RoboDK station: ROBODK_SIGNAL_BOX_V1.rdk

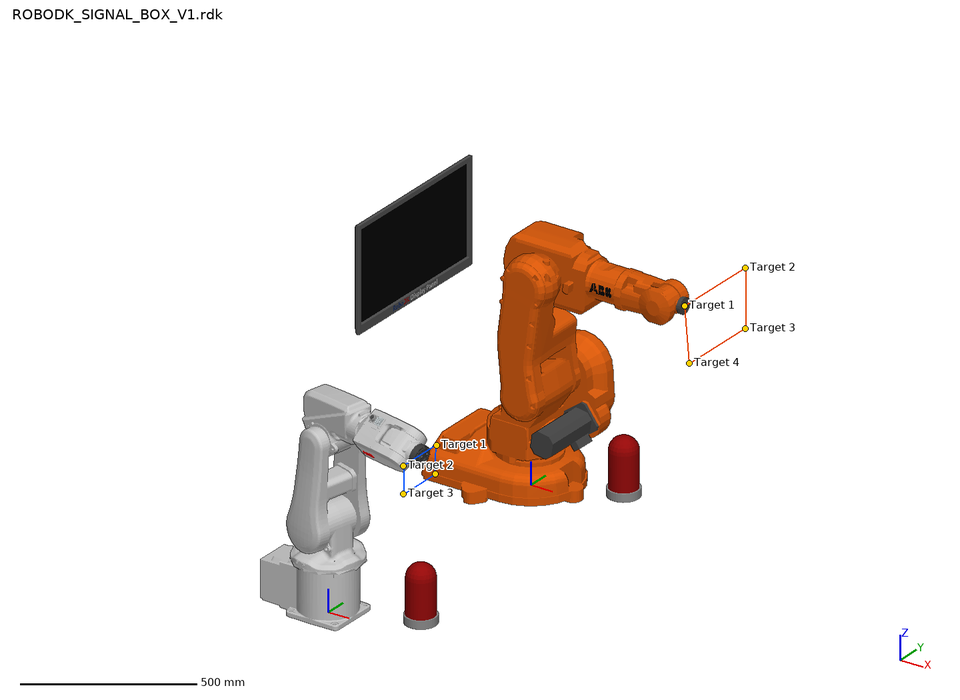
[picture v0: the station drawn from its stored meshes, robots at their saved joint values, targets as dots, program paths as lines]
Station ROBODK 3D PRINT AND CONTROLLER (saved by RoboDK 5.7.4). Poses are relative to the parent item; angles as X-Y-Z fixed-axis rotations.
Station parameters (name, value as stored): IO_1, 0, IO_2, 0, Photodiode, 740
  - frame ABB IRB 120-3/0.6 Base at (0, 0, 0) mm
    - robot ABB IRB 120-3/0.3 (model ABB IRB 120-3/0.6): 6 axes, payload 3 kg, reach 580 mm, repeatability 0.01 mm, weight 25 kg
        modified DH rows (alpha deg, a mm, theta deg, d mm): 0, 0, 0, 290; -90, 0, -90, 0; 0, 270, 0, 0; -90, 70, 0, 302; 90, 0, 0, 0; -90, 0, 180, 72
        joint limits [-165, -110, -90, -160, -120, -400] to [165, 110, 70, 160, 120, 400]; home [0, 0, 0, 0, 0, 0]; saved at [-12.428, 3.919, -4.192, 38.932, 12.431, -38.863]
    - target Target 1 (Cartesian target) at (374, 0, 630) mm, rotated rx 0 ry 90 rz 0 deg; joints [0, 0, 0, 0, 0, 0] of ABB IRB 120-3/0.3
    - target Target 2 (Cartesian target) at (374, -163.03, 630) mm, rotated rx 0 ry 90 rz 0 deg; joints [-28.361, 8.943, -9.567, 88.845, 28.367, -88.688] of ABB IRB 120-3/0.3
    - target Target 3 (Cartesian target) at (374, -163.03, 540.71) mm, rotated rx 0 ry 90 rz 0 deg; joints [-28.361, 7.162, 9.065, 117.369, 32.337, -121.495] of ABB IRB 120-3/0.3
    - target Target 4 (Cartesian target) at (374, -6.94, 540.71) mm, rotated rx 0 ry 90 rz 0 deg; joints [-1.317, -1.556, 18.155, -4.601, -16.65, 4.409] of ABB IRB 120-3/0.3
  - frame ABB IRB 140-6/0.8 Base at (0, 1000, 0) mm
    - robot ABB IRB 140-6/0.8: 6 axes, payload 6 kg, reach 810 mm, repeatability 0.03 mm, weight 98 kg
        modified DH rows (alpha deg, a mm, theta deg, d mm): 0, 0, 0, 352; -90, 70, -90, 0; 0, 360, 0, 0; -90, 0, 0, 380; 90, 0, 0, 0; -90, 0, 180, 65
        joint limits [-180, -90, -230, -200, -120, -400] to [180, 110, 50, 200, 120, 400]; home [0, 0, 0, 0, 0, 0]; saved at [0, 2.547, -2.601, 0, 0.054, 0]
    - target Target 1 (Cartesian target) at (531, 0, 712) mm, rotated rx 0 ry 90 rz 0 deg; joints [0, 2.547, -2.601, 0, 0.054, 0] of ABB IRB 140-6/0.8
    - target Target 2 (Cartesian target) at (531, 299.55, 712) mm, rotated rx 0 ry 90 rz 0 deg; joints [32.733, 16.839, -19.167, -86.384, 32.807, 85.7] of ABB IRB 140-6/0.8
    - target Target 3 (Cartesian target) at (531, 299.55, 521.32) mm, rotated rx 0 ry 90 rz 0 deg; joints [32.733, 22.942, 2.325, -123.585, 40.473, 131.118] of ABB IRB 140-6/0.8
    - target Target 4 (Cartesian target) at (531, 23.54, 521.32) mm, rotated rx 0 ry 90 rz 0 deg; joints [2.892, 10.334, 18.771, -174.07, 29.236, 174.821] of ABB IRB 140-6/0.8
  - program Start rob 1 (7 instructions, listed below)
  - program Start rob 2 (7 instructions, listed below)
  - program SET_IO1_0 (3 instructions, listed below)
  - program SET_IO1_1 (4 instructions, listed below)
  - program SET_IO2_0 (3 instructions, listed below)
  - program SET_IO2_1 (4 instructions, listed below)
  - program SET_PD (1 instructions, listed below)
  - object Light_R1_RED at (250, 100, 0) mm, size 100 x 100 x 185.3 mm, geometry from Light-Red.sld
  - object Light_R2_RED at (250, 1100, 0) mm, size 100 x 100 x 185.3 mm, geometry from Light-Red.sld
  - object Light_R1_GREEN at (250, 100, 0) mm, size 100 x 100 x 185.3 mm, geometry from Light-Red.sld
  - object Light_R2_GREEN at (250, 1100, 0) mm, size 100 x 100 x 185.3 mm, geometry from Light-Red.sld
  - object Display Panel 24in at (0, 400, 1000) mm, size 43 x 556.4 x 342.2 mm, geometry from PLUGIN_DISPLAY_DATAU
  - Python program serial_com_test_1 (listed below)
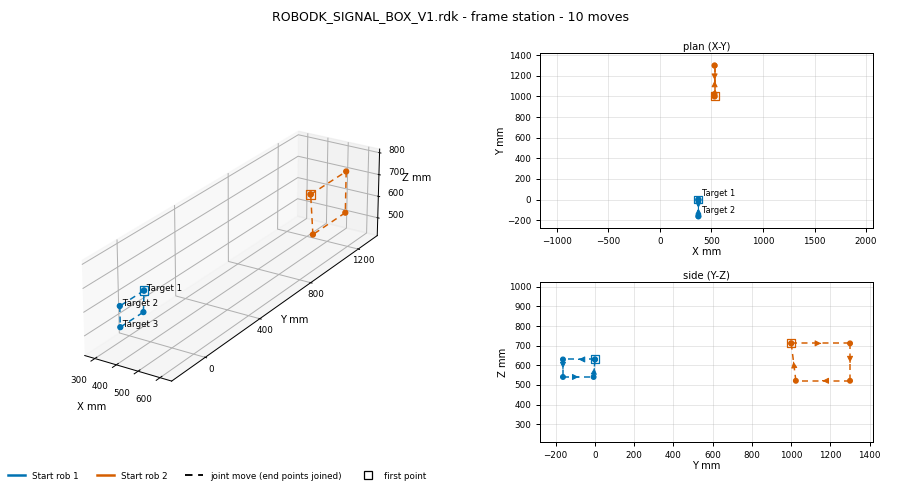
[picture p0: tool path of ROBODK_SIGNAL_BOX_V1.rdk in frame station, 10 of 10 moves have a stored position in this frame; points joined in program order, loops and branches not executed]

--- program Start rob 1 (robot ABB IRB 120-3/0.3) ---
  Set Ref.: ABB IRB 120-3/0.6 Base
  Wait IO_1=1
  MoveJ (Target 1)
  MoveJ (Target 2)
  MoveJ (Target 3)
  MoveJ (Target 4)
  MoveJ (Target 1)

--- program Start rob 2 (robot ABB IRB 140-6/0.8) ---
  Set Ref.: ABB IRB 140-6/0.8 Base
  Wait IO_2=1
  MoveJ (Target 1)
  MoveJ (Target 2)
  MoveJ (Target 3)
  MoveJ (Target 4)
  MoveJ (Target 1)

--- program SET_IO1_0 (robot ABB IRB 120-3/0.3) ---
  Set IO_1=0
  Hide Light_R1_GREEN
  Show Light_R1_RED

--- program SET_IO1_1 (robot ABB IRB 120-3/0.3) ---
  Set IO_1=1
  Show Light_R1_GREEN
  Hide Light_R1_RED
  Call Start rob 1

--- program SET_IO2_0 (robot ABB IRB 120-3/0.3) ---
  Set IO_2=0
  Hide Light_R2_GREEN
  Show Light_R2_RED

--- program SET_IO2_1 (robot ABB IRB 120-3/0.3) ---
  Set IO_2=1
  Hide Light_R2_RED
  Show Light_R2_GREEN
  Call Start rob 2

--- program SET_PD (robot ABB IRB 120-3/0.3) ---
  Set AO_5=1

--- Python program serial_com_test_1 ---
import tkinter as tk
import time
import serial
from robolink import Robolink  # Ensure this is imported correctly
from datetime import datetime  # Import datetime module for formatting the timestamp

# Initialize RoboDK and serial communication
RDK = Robolink()
ser = serial.Serial('COM4', 115200)

# Keep track of previous sensor values
prev_sensor1_value = None
prev_sensor2_value = None

# Log file setup
log_file = "D:/UPB/2024_2025_SEM_1/Articole/01_RoboDK signal Box/documente_articol_v1/latency_log.txt"

# Function to log latency and timestamp
def log_latency(latency, timestamp):
    # Convert timestamp to a readable format
    formatted_time = datetime.fromtimestamp(timestamp).strftime('%Y-%m-%d %H:%M:%S.%f')
    with open(log_file, "a") as file:
        file.write(f"{formatted_time}, {latency:.6f} ms\n")

# Function to handle executing RoboDK programs and updating the UI label
def execute_program_and_update_label(program_name, label):
    RDK.RunProgram(program_name)
    if program_name == "SET_IO1_0":
        label["text"] = "Sensor 1 Value: 0"
        label["bg"] = "yellow"
    elif program_name == "SET_IO1_1":
        label["text"] = "Sensor 1 Value: 1"
        label["bg"] = "green"
    elif program_name == "SET_IO2_0":
        label["text"] = "Sensor 2 Value: 0"
        label["bg"] = "yellow"
    elif program_name == "SET_IO2_1":
        label["text"] = "Sensor 2 Value: 1"
        label["bg"] = "green"

# Function to continuously read data from Arduino and update the UI
def read_arduino_data():
    global prev_sensor1_value, prev_sensor2_value
    while True:
        try:
            # Flush the serial buffer if it's too full
            if ser.in_waiting > 100:
                ser.reset_input_buffer()

            # Start measuring time when data is read
            start_time_pc = time.perf_counter()

            # Read data from Arduino
            if ser.in_waiting > 0:
                data = ser.readline().decode().strip()

                # Split the data into sensor identifier, value, and timestamp
                sensor, value, arduino_timestamp = data.split('_')
                arduino_timestamp = float(arduino_timestamp)

                # Check the current mode (manual/automatic)
                if current_mode.get() == 1:  # Only process Arduino data in automatic mode
                    # Calculate processing time
                    processing_time = (time.perf_counter() - start_time_pc) * 1000  # Convert to ms

                    # Handle IO1 (sensor 1)
                    if sensor == "IO1" and value != prev_sensor1_value:
                        prev_sensor1_value = value
                        execute_program_and_update_label(f"SET_IO1_{value}", label_signal_s1)
                        print(f"Arduino-to-Python processing time: {processing_time:.6f} ms")

                    # Handle IO2 (sensor 2)
                    elif sensor == "IO2" and value != prev_sensor2_value:
                        prev_sensor2_value = value
                        execute_program_and_update_label(f"SET_IO2_{value}", label_signal_s2)
                        print(f"Arduino-to-Python processing time: {processing_time:.6f} ms")

                    # Handle Photodiode (PD) sensor
                    elif sensor == "PD":
                        label_signal_pd["text"] = f"Photodiode Value: {value}"
                        RDK.setParam('Photodiode', value)

                    # End measuring time after running the RoboDK program
                    end_time_pc = time.perf_counter()
                    end_to_end_latency = (end_time_pc - start_time_pc) * 1000  # Convert to ms
                    timestamp = time.time()  # Get the current time in seconds
                    print(f"End-to-End Latency: {end_to_end_latency:.6f} ms")

                     # Log the end-to-end latency and timestamp
                    log_latency(end_to_end_latency, timestamp)

            # Small delay to avoid overwhelming the buffer
            time.sleep(0.01)

        except Exception as e:
            print(f"Error reading Arduino data: {e}")

# Function to handle mode change in the UI (manual/automatic mode)
def change_mode():
    if current_mode.get() == 0:
        label_mode.config(text="Mode: Manual")
        for button in buttons_manual.values():
            button.config(state=tk.NORMAL)
    else:
        label_mode.config(text="Mode: Automatic")
        for button in buttons_manual.values():
            button.config(state=tk.DISABLED)

# Create the main tkinter window
root = tk.Tk()
root.title("RoboDK Control")

# Create Tkinter variable for mode selection
current_mode = tk.IntVar()
current_mode.set(0)  # Initialize mode as manual

# Create labels to display signal values
label_signal_s1 = tk.Label(root, text="Sensor 1 Value: 0", bg="yellow")
label_signal_s1.pack()

label_signal_s2 = tk.Label(root, text="Sensor 2 Value: 0", bg="yellow")
label_signal_s2.pack()

label_signal_pd = tk.Label(root, text="Photodiode Value: 0", bg="yellow")
label_signal_pd.pack()

# Create a label to display the current mode
label_mode = tk.Label(root, text="Mode: Manual")
label_mode.pack()

# Create buttons for program execution in manual mode
buttons_manual = {}
program_names = ["SET_IO1_0", "SET_IO1_1", "SET_IO2_0", "SET_IO2_1"]

for program_name in program_names:
    buttons_manual[program_name] = tk.Button(root, text=program_name,
                                             command=lambda name=program_name: execute_program_and_update_label(name, label_signal_s1 if "IO1" in name else label_signal_s2))
    buttons_manual[program_name].pack()

# Create radio buttons for mode selection
radio_manual = tk.Radiobutton(root, text="Manual", variable=current_mode, value=0, command=change_mode)
radio_manual.pack()

radio_auto = tk.Radiobutton(root, text="Automatic", variable=current_mode, value=1, command=change_mode)
radio_auto.pack()

# Start a thread to continuously read data from Arduino
import threading
arduino_thread = threading.Thread(target=read_arduino_data)
arduino_thread.daemon = True
arduino_thread.start()

# Start the tkinter main loop
root.mainloop()
